(*
    TcXunit interpreter fixture (TcXunit-w5x.8). Base counter: FB_init sets the
    start value, Increment adds, Decrement clamps at a floor read through a
    POINTER TO INT to exercise the v1 pointer/ADR subset.
*)
FUNCTION_BLOCK FB_Counter
VAR
	value : INT;
END_VAR

METHOD PUBLIC Decrement
VAR_INPUT
	delta : INT := 1;
END_VAR
VAR
	floor : INT := 0;
	pFloor : POINTER TO INT;
END_VAR
pFloor := ADR(floor);

IF value - delta < pFloor^ THEN
	value := pFloor^;
ELSE
	value := value - delta;
END_IF
END_METHOD

METHOD FB_init
VAR_INPUT
	bInitRetains : BOOL;
	bInCopyCode : BOOL;
	startValue : INT := 0;
END_VAR
value := startValue;
END_METHOD

METHOD PUBLIC GetValue : INT
GetValue := value;
END_METHOD

METHOD PUBLIC Increment
VAR_INPUT
	delta : INT := 1;
END_VAR
value := value + delta;
END_METHOD

END_FUNCTION_BLOCK

(* stored: Version 1.1.0.1, ProductVersion 3.1.4026.18
   POU FB_Counter: Id {a1b2c3d4-0001-4a1a-8b1b-000000000001}, SpecialFunc None
   Method Decrement: Id {a1b2c3d4-0001-4a1a-8b1b-000000000004}
   Method FB_init: Id {a1b2c3d4-0001-4a1a-8b1b-000000000002}
   Method GetValue: Id {a1b2c3d4-0001-4a1a-8b1b-000000000005}
   Method Increment: Id {a1b2c3d4-0001-4a1a-8b1b-000000000003} *)
